FUNCTION_BLOCK SimpleTestType
  (* Version 1.0, 2005-04-08, Goran Cengic, Chalmers *)
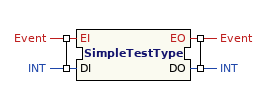
  EVENT_INPUT
    EI WITH DI;
  END_EVENT
  EVENT_OUTPUT
    EO WITH DO;
  END_EVENT
  VAR_INPUT
    DI : INT;
  END_VAR
  VAR_OUTPUT
    DO : INT;
  END_VAR
  VAR
    invoked : INT;
  END_VAR
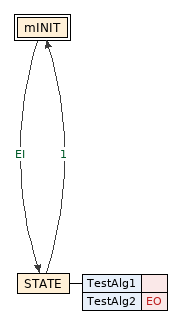
  EC_STATES
    mINIT;
    STATE : TestAlg1, TestAlg2 -> EO;
  END_STATES
  EC_TRANSITIONS
    mINIT TO STATE := EI;
    STATE TO mINIT := 1;
  END_TRANSITIONS
  ALGORITHM TestAlg1 IN Java:
invoked = DI + 1;
	System.out.println("TestAlg1: DI: " + DI + ".");
	System.out.println("TestAlg1:invoked: " + invoked + " times.");
  END_ALGORITHM
  ALGORITHM TestAlg2 IN Java:
DO = invoked + 1;
	System.out.println("TestAlg2:invoked: " + invoked + " times.");
	System.out.println("TestAlg2: DO: " + DO + ".");
  END_ALGORITHM
END_FUNCTION_BLOCK
